FUNCTION SubString
VAR_INPUT
	source : ANY;
	destination : ANY;
	startIndex : DINT;
	length : DINT;
END_VAR
VAR
END_VAR

IF (startIndex >= source.diSize) THEN
	RETURN;
END_IF

MEMCPY(
	destAddr := destination.pValue,
	srcAddr := source.pValue + TO_DWORD(startIndex),
	n := TO_UDINT(MIN(length, MIN(source.diSize - startIndex, destination.diSize)))
);

END_FUNCTION

(* stored: Version 1.1.0.1
   POU SubString: Id {24db83fa-d3af-045a-176e-feaf2ee63db3}, SpecialFunc None *)
